// class for robot units.
FUNCTION_BLOCK Robot EXTENDS UnitBaseClass
VAR_INPUT
	inputMode		:	E_PMLProtectedUnitMode;
	inputCommand	:	E_PMLCommand;
	//inputAxes		:	ST_KinAxes;
END_VAR
VAR_OUTPUT
	pos		:	E6POS;
END_VAR
VAR
	//axes	:	ST_KinAxes;
END_VAR

IF NOT initialized THEN
	SUPER^(modeCommand:=inputMode, command:=inputCommand);
	// axes := inputAxes;
END_IF

METHOD fkine : BOOL
VAR_INPUT
END_VAR
END_METHOD

METHOD ikine : BOOL
VAR_INPUT
END_VAR
END_METHOD

METHOD moveFree : BOOL
VAR_INPUT
END_VAR
END_METHOD

METHOD moveLinear : BOOL
VAR_INPUT
END_VAR
END_METHOD

END_FUNCTION_BLOCK

(* stored: Version 1.1.0.1, ProductVersion 3.1.4022.16
   POU Robot: Id {4157a4ec-321e-422b-a1d1-68c974b07a39}, SpecialFunc None
   Method fkine: Id {fdeeb45d-ca6e-4d23-9004-40bbb1bd3b18}
   Method ikine: Id {2381d57d-ea26-4bd9-9cbe-9a28e869140f}
   Method moveFree: Id {8aa14a30-984d-425d-8468-eb4cf31a65dd}
   Method moveLinear: Id {f6f4b16f-ceac-4e73-a5da-a4bc7eee3a64} *)
